KUKA KRL program: MFORCETEST1.src, MFORCETEST1.dat

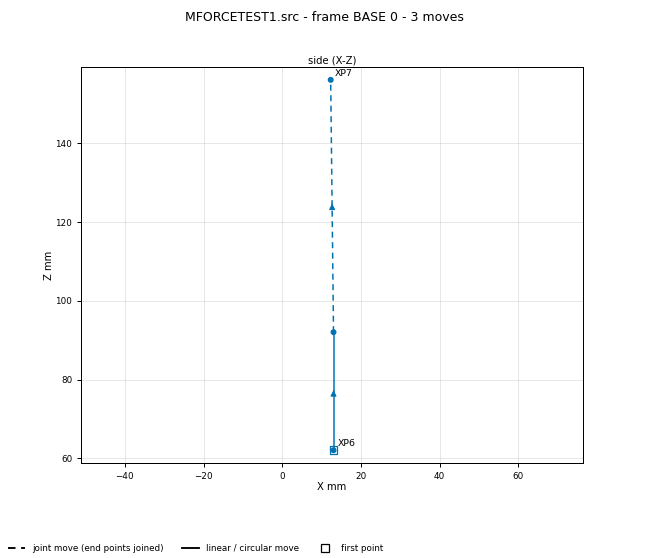
[picture p0: tool path of MFORCETEST1.src in frame BASE 0, 3 of 3 moves have a stored position in this frame; points joined in program order, loops and branches not executed]
--- MFORCETEST1.src ---
&ACCESS RVP
&REL 74
&PARAM TEMPLATE = C:\KRC\Roboter\Template\vorgabe
&PARAM EDITMASK = *
DEF MFORCETEST1( )

INT X
DECL BOOL TEMP, SEMP, HEMP, REMP
DECL E6AXIS TORQUE
REAL PERCENT, STEP

;FOLD INI
  ;FOLD BASISTECH INI
    GLOBAL INTERRUPT DECL 3 WHEN $STOPMESS==TRUE DO IR_STOPM ( )
    INTERRUPT ON 3
    BAS (#INITMOV,0 )
  ;ENDFOLD (BASISTECH INI)
  ;FOLD USER INI
    ;Make your modifications here
  ;ENDFOLD (USER INI)
;ENDFOLD (INI)

$TOOL=TOOL_DATA[5]
FOR X=1 TO 6
$ACC_AXIS[X]=100
$VEL_AXIS[X]=100
ENDFOR

$OV_PRO=100

;FOLD PTP P6 Vel=100 % PDAT6 Tool[5]:Pneumatic_gripper_probe Base[0];%{PE}%R 5.6.11,%MKUKATPBASIS,%CMOVE,%VPTP,%P 1:PTP, 2:P6, 3:, 5:100, 7:PDAT6
$BWDSTART=FALSE
PDAT_ACT=PPDAT6
FDAT_ACT=FP6
BAS(#PTP_PARAMS,100)
PTP XP6
;ENDFOLD



TORQUE=$TORQUE_AXIS_ACT

REMP=FALSE
PERCENT=.5
STEP=-.1

WHILE NOT REMP
  LIN_REL{Z -.1}
  TORQUE=$TORQUE_AXIS_ACT
  REMP=TORQUE.A1>(176*PERCENT)
  REMP= REMP OR (ABS(TORQUE.A2)>(176*PERCENT))
  REMP= REMP OR (ABS(TORQUE.A3)>(100*PERCENT))
  REMP= REMP OR (ABS(TORQUE.A4)>(100*PERCENT))
  REMP= REMP OR (ABS(TORQUE.A5)>(38*PERCENT))
  REMP= REMP OR (ABS(TORQUE.A6)>(38*PERCENT))
ENDWHILE

LIN_REL {Z 30}

;FOLD PTP P7 Vel=100 % PDAT7 Tool[5]:Pneumatic_gripper_probe Base[0];%{PE}%R 5.6.11,%MKUKATPBASIS,%CMOVE,%VPTP,%P 1:PTP, 2:P7, 3:, 5:100, 7:PDAT7
$BWDSTART=FALSE
PDAT_ACT=PPDAT7
FDAT_ACT=FP7
BAS(#PTP_PARAMS,100)
PTP XP7
;ENDFOLD


END

--- MFORCETEST1.dat ---
&ACCESS RVP
&REL 74
&PARAM TEMPLATE = C:\KRC\Roboter\Template\vorgabe
&PARAM EDITMASK = *
DEFDAT  MFORCETEST1
;FOLD EXTERNAL DECLARATIONS;%{PE}%MKUKATPBASIS,%CEXT,%VCOMMON,%P
;FOLD BASISTECH EXT;%{PE}%MKUKATPBASIS,%CEXT,%VEXT,%P
EXT  BAS (BAS_COMMAND  :IN,REAL  :IN )
DECL INT SUCCESS
;ENDFOLD (BASISTECH EXT)
;FOLD USER EXT;%{E}%MKUKATPUSER,%CEXT,%VEXT,%P
;Make here your modifications

;ENDFOLD (USER EXT)
;ENDFOLD (EXTERNAL DECLARATIONS)
DECL BASIS_SUGG_T LAST_BASIS={POINT1[] "P7                      ",POINT2[] "P7                      ",CP_PARAMS[] "CPDAT0                  ",PTP_PARAMS[] "PDAT7                   ",CONT[] "                        ",CP_VEL[] "2.0                     ",PTP_VEL[] "100                     ",SYNC_PARAMS[] "SYNCDAT                 ",SPL_NAME[] "S0                      "}
DECL PDAT PPDAT0={VEL 100.0,ACC 100.0,APO_DIST 100.0,APO_MODE #CPTP}
DECL E6POS XP0={X 12.30126,Y -591.60022,Z 156.144394,A 1.17926598,B -0.00117073196,C -179.9776,S 1,T 36,E1 -0.0129604302,E2 0.0,E3 0.0,E4 0.0,E5 0.0,E6 0.0}
DECL FDAT FP0={TOOL_NO 5,BASE_NO 0,IPO_FRAME #BASE,POINT2[] " ",TQ_STATE FALSE}
DECL PDAT PPDAT1={VEL 100.0,ACC 100.0,APO_DIST 100.0,APO_MODE #CPTP}
DECL E6POS XP1={X 12.30126,Y -591.60022,Z 156.144394,A 1.17926598,B -0.00117073196,C -179.9776,S 1,T 36,E1 -0.0129604302,E2 0.0,E3 0.0,E4 0.0,E5 0.0,E6 0.0}
DECL FDAT FP1={TOOL_NO 5,BASE_NO 0,IPO_FRAME #BASE,POINT2[] " ",TQ_STATE FALSE}
DECL PDAT PPDAT2={VEL 100.0,ACC 100.0,APO_DIST 100.0,APO_MODE #CPTP}
DECL E6POS XP2={X 12.30126,Y -591.60022,Z 156.144394,A 1.17926598,B -0.00117073196,C -179.9776,S 1,T 36,E1 -0.0129604302,E2 0.0,E3 0.0,E4 0.0,E5 0.0,E6 0.0}
DECL FDAT FP2={TOOL_NO 5,BASE_NO 0,IPO_FRAME #BASE,POINT2[] " ",TQ_STATE FALSE}
DECL PDAT PPDAT3={VEL 100.0,ACC 100.0,APO_DIST 100.0,APO_MODE #CPTP}
DECL E6POS XP3={X 12.30126,Y -591.60022,Z 156.144394,A 1.17926598,B -0.00117073196,C -179.9776,S 1,T 36,E1 -0.0129604302,E2 0.0,E3 0.0,E4 0.0,E5 0.0,E6 0.0}
DECL FDAT FP3={TOOL_NO 5,BASE_NO 0,IPO_FRAME #BASE,POINT2[] " ",TQ_STATE FALSE}
DECL PDAT PPDAT4={VEL 100.0,ACC 100.0,APO_DIST 100.0,APO_MODE #CPTP}
DECL E6POS XP4={X 12.30126,Y -591.60022,Z 156.144394,A 1.17926598,B -0.00117073196,C -179.9776,S 1,T 36,E1 -0.0129604302,E2 0.0,E3 0.0,E4 0.0,E5 0.0,E6 0.0}
DECL FDAT FP4={TOOL_NO 5,BASE_NO 0,IPO_FRAME #BASE,POINT2[] " ",TQ_STATE FALSE}
DECL PDAT PPDAT5={VEL 100.0,ACC 100.0,APO_DIST 100.0,APO_MODE #CPTP}
DECL E6POS XP5={X 12.30126,Y -591.60022,Z 156.144394,A 1.17926598,B -0.00117073196,C -179.9776,S 1,T 36,E1 -0.0129604302,E2 0.0,E3 0.0,E4 0.0,E5 0.0,E6 0.0}
DECL FDAT FP5={TOOL_NO 5,BASE_NO 0,IPO_FRAME #BASE,POINT2[] " ",TQ_STATE FALSE}
DECL PDAT PPDAT6={VEL 100.0,ACC 100.0,APO_DIST 100.0,APO_MODE #CPTP}
DECL E6POS XP6={X 13.0194798,Y -591.27002,Z 62.0346718,A 1.20812094,B -0.0206202809,C -179.929596,S 1,T 36,E1 -0.0109777497,E2 0.0,E3 0.0,E4 0.0,E5 0.0,E6 0.0}
DECL FDAT FP6={TOOL_NO 5,BASE_NO 0,IPO_FRAME #BASE,POINT2[] " ",TQ_STATE FALSE}
DECL PDAT PPDAT7={VEL 100.0,ACC 100.0,APO_DIST 100.0,APO_MODE #CPTP}
DECL E6POS XP7={X 12.30126,Y -591.60022,Z 156.144394,A 1.17926598,B -0.00117073196,C -179.9776,S 1,T 36,E1 -0.0129604302,E2 0.0,E3 0.0,E4 0.0,E5 0.0,E6 0.0}
DECL FDAT FP7={TOOL_NO 5,BASE_NO 0,IPO_FRAME #BASE,POINT2[] " ",TQ_STATE FALSE}
ENDDAT
